(* IEC 61131-3 sources: repolevel_ST_code_completion/dataset/generation_context_ground_truth/Decorator_Application, 14 files *)

(* ---- ConcreteComponment.st ---- *)
VAR
	//String field to store the description of the object
	sDescription : STRING;
	//Real field to store the value of the object
	rValue : REAL;
END_VAR

(* ---- ConcreteComponment_fb_init.st ---- *)
VAR
	//String field to store the description of the object
	sDescription : STRING;
	//Real field to store the value of the object
	rValue : REAL;
END_VAR

//Sets the default description for the objects of this class
THIS^.sDescription := 'Plain Component';
//Sets the default value for the objects of this class
THIS^.rValue := 4.0;

(* ---- ConcreteComponment_getDescription.st ---- *)
VAR
	//String field to store the description of the object
	sDescription : STRING;
	//Real field to store the value of the object
	rValue : REAL;
END_VAR

//Description of the plain object is given
getDescription := This^.sDescription;

(* ---- ConcreteComponment_getValue.st ---- *)
VAR
	//String field to store the description of the object
	sDescription : STRING;
	//Real field to store the value of the object
	rValue : REAL;
END_VAR

//Assume we are going to calculate the cost os the object.
//The plain value (without extra decoration) is given
getValue := THIS^.rValue;

(* ---- ConcreteDecoratorA.st ---- *)
VAR
END_VAR

(* ---- ConcreteDecoratorB.st ---- *)
VAR
END_VAR

(* ---- ConcreteDecoratorB_getDescription.st ---- *)
VAR
END_VAR

//Outputs the decorated description of the component by obtaining the description of the component
// to be decorated stored in tempComponet.getDescription() and then concatenates the decoration
// description( ' Decorator B' as example)
getDescription :=CONCAT(THIS^.tempComponent.getDescription() , THIS^.sDescription);

(* ---- ConcreteDecoratorB_getValue.st ---- *)
VAR
END_VAR

//Outputs the decorated cost of the component by obtaining the cost of the component to be decorated
// stored in tempComponent.getValue() and then adds the decoration value (0.35 as example)
getValue := tempComponent.getValue() + THIS^.rValue;

(* ---- ConcreteDecoratorC.st ---- *)
VAR
END_VAR

(* ---- ConcreteDecoratorC_getDescription.st ---- *)
VAR
END_VAR

//Outputs the decorated description of the component by obtaining the description of the component
// to be decorated stored in tempComponet.getDescription() and then concatenates the decoration
// description( ' Decorator C' as example)
getDescription :=CONCAT(THIS^.tempComponent.getDescription() , THIS^.sDescription);

(* ---- ConcreteDecoratorC_getValue.st ---- *)
VAR
END_VAR

//Outputs the decorated cost of the component by obtaining the cost of the component to be decorated
// stored in tempComponent.getValue() and then adds the decoration value (0.15 as example)
getValue := tempComponent.getValue() + THIS^.rValue;

(* ---- Decorator.st ---- *)
VAR
	//Variable to save the state of the concrete component to be decorated
	tempComponent : Component_Interface;
	//String variable to save the Description of the component
	sDescription : STRING;
	//Real variable to save the Value of the component
	rValue : REAL;
END_VAR

(* ---- Decorator_getDescription.st ---- *)
VAR
	//Variable to save the state of the concrete component to be decorated
	tempComponent : Component_Interface;
	//String variable to save the Description of the component
	sDescription : STRING;
	//Real variable to save the Value of the component
	rValue : REAL;
END_VAR

//Outputs the description of the component to be decorated tempComponent. If tempComponent is not an undecorated component (plain object)
// it means the program has to do at least 2 decorations. Then is going to output the previous decoration complete description
// to be used by the next decorator.
getDescription := THIS^.tempComponent.getDescription();

(* ---- Decorator_getValue.st ---- *)
VAR
	//Variable to save the state of the concrete component to be decorated
	tempComponent : Component_Interface;
	//String variable to save the Description of the component
	sDescription : STRING;
	//Real variable to save the Value of the component
	rValue : REAL;
END_VAR

//Outputs the cost of the component to be decorated tempComponent. If tempComponent is not an undecorated component (plain object)
// it means the program has to do at least 2 decorations. Then is going to output the previous decoration complete value
// to be used by the next decorator.
getValue := tempComponent.getValue();
